# EPICS SNL sequencer program: siteApps/SCL3Cooldown-sim-2-O/cooldownApp/src/CDOM15HWR_2_3.stt
program CDOM15HWR23Logic
option +r;

%% #include <math.h>

int om15HWR23LogicProc[1];
assign om15HWR23LogicProc to {
":CDLogic.PROC"
};
monitor om15HWR23LogicProc;

float valveVal[1];
assign valveVal to {
":Valve"
};

monitor valveVal;

evflag  evFanout;
sync	valveVal	evFanout;

int index = 0;
assign index to "SCL3:CD-OM15HWR23:IndexPV";
monitor index;

int proc = 1;

float om15HWR23Val;
assign om15HWR23Val to "SCL3:CD-OM15HWR23:Value";
monitor om15HWR23Val;

float cdDelay;
assign cdDelay to "SCL3:CD-OM15HWR23:ScanTime";
monitor cdDelay;

float	valvewave[1];
assign	valvewave to "SCL3:CD-OM15HWR23:ValveWave";
monitor valvewave;

ss ssCDOM15HWR23
{
	state CDOM15HWR23
	{
		when(delay(cdDelay))
		{
			if(index == 0  || index == 1  || index == 8  || index == 10 ||
			   index == 12 || index == 14 || index == 16 || index == 18 || index == 20 ||
			   index == 22 || index == 24 || index == 26 || index == 28 || index == 30 ||
			   index == 32 || index == 34 || index == 36 || index == 38 || index == 40 ||
			   index == 42 || index == 44 || index == 46 || index == 48 || index == 50 ||
			   index == 52 || index == 54 || index == 56 || index == 58 || index == 60 ||
			   index == 62 || index == 64 || index == 66 || index == 68 || index == 70 ||
			   index == 72 || index == 75 || index == 78 || index == 81 || index == 84 ||
			   index == 87 || index == 90 || index == 93 || index == 96 || index == 99 ||
			   index == 102|| index == 105)
			{
				if(om15HWR23Val == 1) {
					om15HWR23Val = 0;
					index++;
					pvPut(index, SYNC);
				} else {
					om15HWR23Val = valveVal[index];
				};
			}
			else
			{
				if(om15HWR23Val == 100) {
					om15HWR23Val = 0;
					index++;
					pvPut(index, SYNC);
				} else {
					om15HWR23Val = valveVal[index];
				};
			};

			pvPut(om15HWR23Val, SYNC);
			if(index < 107)
			{
				om15HWR23LogicProc[index] = proc;
				pvPut(om15HWR23LogicProc[index], SYNC);
			};
		}state CDOM15HWR23
	}

}

ss ssOM15HWR23ValveWave
{
	state init
	{
		when(TRUE)
		{
			efClear(evFanout);
		}state MakeOM15HWR23ValveWave
	}

	state MakeOM15HWR23ValveWave
	{
		when(efTestAndClear(evFanout))
		{
			int idx = 0;
			%%for(idx = 0; idx < 107;idx++)
				valvewave[idx] = valveVal[idx];

			pvPut(valvewave, SYNC);
		}state MakeOM15HWR23ValveWave
	}
}
